// Mitsubishi GX Works2 project: PLC_센서_실린더   PLC: Q03UD

PROGRAM MAIN
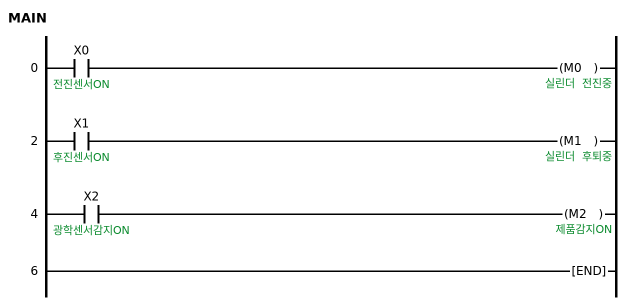
0     LD      X0  ; 전진센서ON
      OUT     M0  ; 실린더  전진중
2     LD      X1  ; 후진센서ON
      OUT     M1  ; 실린더  후퇴중
4     LD      X2  ; 광학센서감지ON
      OUT     M2  ; 제품감지ON
6     END
END_PROGRAM

PROGRAM EX01
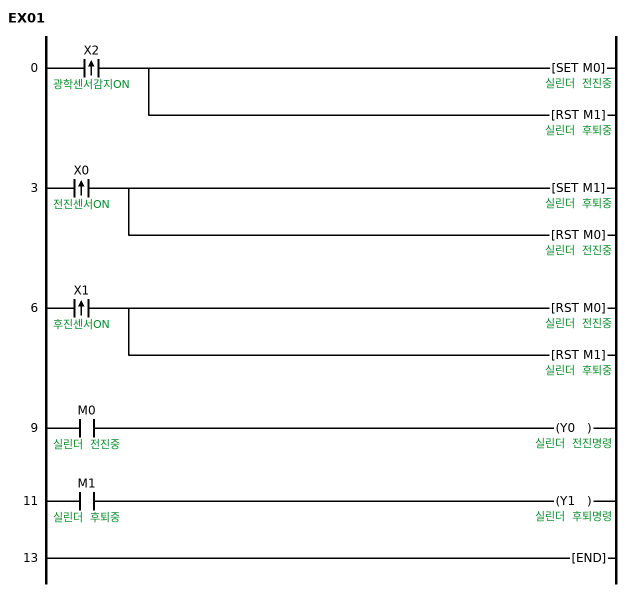
0     LDP     X2  ; 광학센서감지ON
      SET     M0  ; 실린더  전진중
      RST     M1  ; 실린더  후퇴중
3     LDP     X0  ; 전진센서ON
      SET     M1  ; 실린더  후퇴중
      RST     M0  ; 실린더  전진중
6     LDP     X1  ; 후진센서ON
      RST     M0  ; 실린더  전진중
      RST     M1  ; 실린더  후퇴중
9     LD      M0  ; 실린더  전진중
      OUT     Y0  ; 실린더  전진명령
11    LD      M1  ; 실린더  후퇴중
      OUT     Y1  ; 실린더  후퇴명령
13    END
END_PROGRAM
